FUNCTION_BLOCK Load2Check (* Template for a Basic Function Block Type *)
  (* Standard: 61499-2 *)
  (* Version 1.0, 2021-07-28, Tuojian Lyu *)
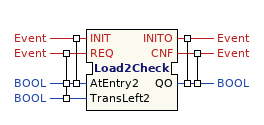
  EVENT_INPUT
    INIT WITH AtEntry2; (* Initialization Request *)
    REQ WITH AtEntry2, TransLeft2; (* Normal Execution Request *)
  END_EVENT
  EVENT_OUTPUT
    INITO WITH QO; (* Initialization Confirm *)
    CNF WITH QO; (* Execution Confirmation *)
  END_EVENT
  VAR_INPUT
    AtEntry2 : BOOL; (* Input event qualifier *)
    TransLeft2 : BOOL;
  END_VAR
  VAR_OUTPUT
    QO : BOOL; (* Output event qualifier *)
  END_VAR
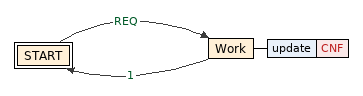
  EC_STATES
    START; (* Initial State *)
    Work : update -> CNF;
  END_STATES
  EC_TRANSITIONS
    START TO Work := REQ;
    Work TO START := 1;
  END_TRANSITIONS
  ALGORITHM update IN ST:
IF (TRUE = AtEntry2) AND (NOT TransLeft2) THEN
QO := TRUE;
ELSE
QO := FALSE;
END_IF;
  END_ALGORITHM
END_FUNCTION_BLOCK
